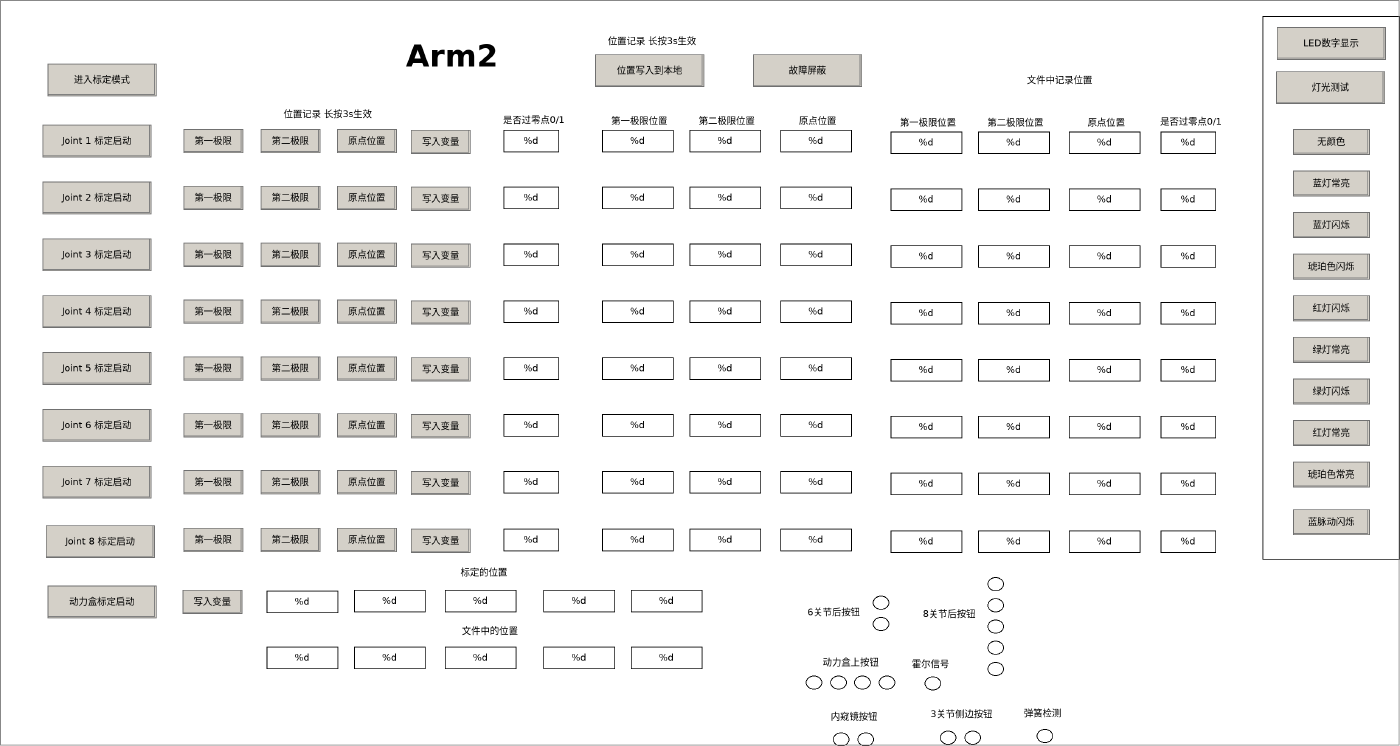
VISUALIZATION arm2Cail  // 1649x879
    Button (56,75 128x38), "进入标定模式", colour toggle: GVL_armCali.g_armEnterCaliMode[2]
        toggle GVL_armCali.g_armEnterCaliMode[2]
    Button (50,147 128x38), "Joint 1 标定启动", colour toggle: GVL_armCali.g_jointIntoCaliState[2][1]
        toggle GVL_armCali.g_jointIntoCaliState[2][1]
    Label (434,40 197x52), "Arm2"
    Button (50,214 128x38), "Joint 2 标定启动", colour toggle: GVL_armCali.g_jointIntoCaliState[2][2]
        toggle GVL_armCali.g_jointIntoCaliState[2][2]
    Button (216,152 70x28), "第一极限", colour toggle: GVL_armCali.g_linkEncFristCaliTrigger[2][1]
        tap GVL_armCali.g_linkEncFristPosCali[2][1]
    Button (307,152 70x28), "第二极限", colour toggle: GVL_armCali.g_linkEncSecondCaliTrigger[2][1]
        tap GVL_armCali.g_linkEncSecondPosCali[2][1]
    Rectangle (593,153 65x26), "%d", text variable: GVL_armCali.g_linkZeroCrossOrNot[2][1]
    Label (588,130 82x23), "是否过零点0/1"
    Rectangle (709,153 84x26), "%d", text variable: GVL_armCali.g_linkLimitFristPos[2][1]
    Label (712,131 82x23), "第一极限位置"
    Rectangle (812,153 84x26), "%d", text variable: GVL_armCali.g_linkLimitSecondPos[2][1]
    Label (815,131 82x23), "第二极限位置"
    Label (311,123 150x23), "位置记录 长按3s生效"
    Rectangle (919,153 84x26), "%d", text variable: GVL_armCali.g_linkHomePos[2][1]
    Label (922,131 82x23), "原点位置"
    Button (397,152 70x28), "原点位置", colour toggle: GVL_armCali.g_linkEncHomePosCaliTrigger[2][1]
        tap GVL_armCali.g_linkEncHomePosCali[2][1]
    Button (701,64 128x38), "位置写入到本地", colour toggle: GVL_armCali.g_caliDataWriteTrigger[2]
        tap GVL_armCali.g_caliDataWrite[2]
    Label (693,37 150x23), "位置记录 长按3s生效"
    Button (216,219 70x28), "第一极限", colour toggle: GVL_armCali.g_linkEncFristCaliTrigger[2][2]
        tap GVL_armCali.g_linkEncFristPosCali[2][2]
    Button (307,219 70x28), "第二极限", colour toggle: GVL_armCali.g_linkEncSecondCaliTrigger[2][2]
        tap GVL_armCali.g_linkEncSecondPosCali[2][2]
    Rectangle (593,220 65x26), "%d", text variable: GVL_armCali.g_linkZeroCrossOrNot[2][2]
    Rectangle (709,220 84x26), "%d", text variable: GVL_armCali.g_linkLimitFristPos[2][2]
    Rectangle (812,220 84x26), "%d", text variable: GVL_armCali.g_linkLimitSecondPos[2][2]
    Rectangle (919,220 84x26), "%d", text variable: GVL_armCali.g_linkHomePos[2][2]
    Button (397,219 70x28), "原点位置", colour toggle: GVL_armCali.g_linkEncHomePosCaliTrigger[2][2]
        tap GVL_armCali.g_linkEncHomePosCali[2][2]
    Button (50,281 128x38), "Joint 3 标定启动", colour toggle: GVL_armCali.g_jointIntoCaliState[2][3]
        toggle GVL_armCali.g_jointIntoCaliState[2][3]
    Button (216,286 70x28), "第一极限", colour toggle: GVL_armCali.g_linkEncFristCaliTrigger[2][3]
        tap GVL_armCali.g_linkEncFristPosCali[2][3]
    Button (307,286 70x28), "第二极限", colour toggle: GVL_armCali.g_linkEncSecondCaliTrigger[2][3]
        tap GVL_armCali.g_linkEncSecondPosCali[2][3]
    Rectangle (593,287 65x26), "%d", text variable: GVL_armCali.g_linkZeroCrossOrNot[2][3]
    Rectangle (709,287 84x26), "%d", text variable: GVL_armCali.g_linkLimitFristPos[2][3]
    Rectangle (812,287 84x26), "%d", text variable: GVL_armCali.g_linkLimitSecondPos[2][3]
    Rectangle (919,287 84x26), "%d", text variable: GVL_armCali.g_linkHomePos[2][3]
    Button (397,286 70x28), "原点位置", colour toggle: GVL_armCali.g_linkEncHomePosCaliTrigger[2][3]
        tap GVL_armCali.g_linkEncHomePosCali[2][3]
    Button (50,348 128x38), "Joint 4 标定启动", colour toggle: GVL_armCali.g_jointIntoCaliState[2][4]
        toggle GVL_armCali.g_jointIntoCaliState[2][4]
    Button (216,353 70x28), "第一极限", colour toggle: GVL_armCali.g_linkEncFristCaliTrigger[2][4]
        tap GVL_armCali.g_linkEncFristPosCali[2][4]
    Button (307,353 70x28), "第二极限", colour toggle: GVL_armCali.g_linkEncSecondCaliTrigger[2][4]
        tap GVL_armCali.g_linkEncSecondPosCali[2][4]
    Rectangle (593,354 65x26), "%d", text variable: GVL_armCali.g_linkZeroCrossOrNot[2][4]
    Rectangle (709,354 84x26), "%d", text variable: GVL_armCali.g_linkLimitFristPos[2][4]
    Rectangle (812,354 84x26), "%d", text variable: GVL_armCali.g_linkLimitSecondPos[2][4]
    Rectangle (919,354 84x26), "%d", text variable: GVL_armCali.g_linkHomePos[2][4]
    Button (397,353 70x28), "原点位置", colour toggle: GVL_armCali.g_linkEncHomePosCaliTrigger[2][4]
        tap GVL_armCali.g_linkEncHomePosCali[2][4]
    Button (50,415 128x38), "Joint 5 标定启动", colour toggle: GVL_armCali.g_jointIntoCaliState[2][5]
        toggle GVL_armCali.g_jointIntoCaliState[2][5]
    Button (216,420 70x28), "第一极限", colour toggle: GVL_armCali.g_linkEncFristCaliTrigger[2][5]
        tap GVL_armCali.g_linkEncFristPosCali[2][5]
    Button (307,420 70x28), "第二极限", colour toggle: GVL_armCali.g_linkEncSecondCaliTrigger[2][5]
        tap GVL_armCali.g_linkEncSecondPosCali[2][5]
    Rectangle (593,421 65x26), "%d", text variable: GVL_armCali.g_linkZeroCrossOrNot[2][5]
    Rectangle (709,421 84x26), "%d", text variable: GVL_armCali.g_linkLimitFristPos[2][5]
    Rectangle (812,421 84x26), "%d", text variable: GVL_armCali.g_linkLimitSecondPos[2][5]
    Rectangle (919,421 84x26), "%d", text variable: GVL_armCali.g_linkHomePos[2][5]
    Button (397,420 70x28), "原点位置", colour toggle: GVL_armCali.g_linkEncHomePosCaliTrigger[2][5]
        tap GVL_armCali.g_linkEncHomePosCali[2][5]
    Button (50,482 128x38), "Joint 6 标定启动", colour toggle: GVL_armCali.g_jointIntoCaliState[2][6]
        toggle GVL_armCali.g_jointIntoCaliState[2][6]
    Button (216,487 70x28), "第一极限", colour toggle: GVL_armCali.g_linkEncFristCaliTrigger[2][6]
        tap GVL_armCali.g_linkEncFristPosCali[2][6]
    Button (307,487 70x28), "第二极限", colour toggle: GVL_armCali.g_linkEncSecondCaliTrigger[2][6]
        tap GVL_armCali.g_linkEncSecondPosCali[2][6]
    Rectangle (593,488 65x26), "%d", text variable: GVL_armCali.g_linkZeroCrossOrNot[2][6]
    Rectangle (709,488 84x26), "%d", text variable: GVL_armCali.g_linkLimitFristPos[2][6]
    Rectangle (812,488 84x26), "%d", text variable: GVL_armCali.g_linkLimitSecondPos[2][6]
    Rectangle (919,488 84x26), "%d", text variable: GVL_armCali.g_linkHomePos[2][6]
    Button (397,487 70x28), "原点位置", colour toggle: GVL_armCali.g_linkEncHomePosCaliTrigger[2][6]
        tap GVL_armCali.g_linkEncHomePosCali[2][6]
    Button (50,549 128x38), "Joint 7 标定启动", colour toggle: GVL_armCali.g_jointIntoCaliState[2][7]
        toggle GVL_armCali.g_jointIntoCaliState[2][7]
    Button (216,554 70x28), "第一极限", colour toggle: GVL_armCali.g_linkEncFristCaliTrigger[2][7]
        tap GVL_armCali.g_linkEncFristPosCali[2][7]
    Button (307,554 70x28), "第二极限", colour toggle: GVL_armCali.g_linkEncSecondCaliTrigger[2][7]
        tap GVL_armCali.g_linkEncSecondPosCali[2][7]
    Rectangle (593,555 65x26), "%d", text variable: GVL_armCali.g_linkZeroCrossOrNot[2][7]
    Rectangle (709,555 84x26), "%d", text variable: GVL_armCali.g_linkLimitFristPos[2][7]
    Rectangle (812,555 84x26), "%d", text variable: GVL_armCali.g_linkLimitSecondPos[2][7]
    Rectangle (919,555 84x26), "%d", text variable: GVL_armCali.g_linkHomePos[2][7]
    Button (397,554 70x28), "原点位置", colour toggle: GVL_armCali.g_linkEncHomePosCaliTrigger[2][7]
        tap GVL_armCali.g_linkEncHomePosCali[2][7]
    Button (54,619 128x38), "Joint 8 标定启动", colour toggle: GVL_armCali.g_jointIntoCaliState[2][8]
        toggle GVL_armCali.g_jointIntoCaliState[2][8]
    Button (216,622 70x28), "第一极限", colour toggle: GVL_armCali.g_linkEncFristCaliTrigger[2][8]
        tap GVL_armCali.g_linkEncFristPosCali[2][8]
    Button (307,622 70x28), "第二极限", colour toggle: GVL_armCali.g_linkEncSecondCaliTrigger[2][8]
        tap GVL_armCali.g_linkEncSecondPosCali[2][8]
    Rectangle (593,623 65x26), "%d", text variable: GVL_armCali.g_linkZeroCrossOrNot[2][8]
    Rectangle (709,623 84x26), "%d", text variable: GVL_armCali.g_linkLimitFristPos[2][8]
    Rectangle (812,623 84x26), "%d", text variable: GVL_armCali.g_linkLimitSecondPos[2][8]
    Rectangle (919,623 84x26), "%d", text variable: GVL_armCali.g_linkHomePos[2][8]
    Button (397,622 70x28), "原点位置", colour toggle: GVL_armCali.g_linkEncHomePosCaliTrigger[2][8]
        tap GVL_armCali.g_linkEncHomePosCali[2][8]
    Rectangle (1049,155 84x26), "%d", text variable: GVL_SetupJointEncoderCaliData.g_minLinkEncoder[2,1]
    Label (1052,133 82x23), "第一极限位置"
    Rectangle (1152,155 84x26), "%d", text variable: GVL_SetupJointEncoderCaliData.g_maxLinkEncoder[2,1]
    Label (1155,133 82x23), "第二极限位置"
    Rectangle (1259,155 84x26), "%d", text variable: GVL_SetupJointEncoderCaliData.g_caliLinkEncoder[2,1]
    Label (1262,133 82x23), "原点位置"
    Rectangle (1049,222 84x26), "%d", text variable: GVL_SetupJointEncoderCaliData.g_minLinkEncoder[2,2]
    Rectangle (1152,222 84x26), "%d", text variable: GVL_SetupJointEncoderCaliData.g_maxLinkEncoder[2,2]
    Rectangle (1259,222 84x26), "%d", text variable: GVL_SetupJointEncoderCaliData.g_caliLinkEncoder[2,2]
    Rectangle (1049,289 84x26), "%d", text variable: GVL_SetupJointEncoderCaliData.g_minLinkEncoder[2,3]
    Rectangle (1152,289 84x26), "%d", text variable: GVL_SetupJointEncoderCaliData.g_maxLinkEncoder[2,3]
    Rectangle (1259,289 84x26), "%d", text variable: GVL_SetupJointEncoderCaliData.g_caliLinkEncoder[2,3]
    Rectangle (1049,356 84x26), "%d", text variable: GVL_SetupJointEncoderCaliData.g_minLinkEncoder[2,4]
    Rectangle (1152,356 84x26), "%d", text variable: GVL_SetupJointEncoderCaliData.g_maxLinkEncoder[2,4]
    Rectangle (1259,356 84x26), "%d", text variable: GVL_SetupJointEncoderCaliData.g_caliLinkEncoder[2,4]
    Rectangle (1049,423 84x26), "%d", text variable: GVL_SetupJointEncoderCaliData.g_minLinkEncoder[2,5]
    Rectangle (1152,423 84x26), "%d", text variable: GVL_SetupJointEncoderCaliData.g_maxLinkEncoder[2,5]
    Rectangle (1259,423 84x26), "%d", text variable: GVL_SetupJointEncoderCaliData.g_caliLinkEncoder[2,5]
    Rectangle (1049,490 84x26), "%d", text variable: GVL_SlaveJointEncoderCaliData.g_minLinkEncoder[2,1]
    Rectangle (1152,490 84x26), "%d", text variable: GVL_SlaveJointEncoderCaliData.g_maxLinkEncoder[2,1]
    Rectangle (1259,490 84x26), "%d", text variable: GVL_SlaveJointEncoderCaliData.g_caliLinkEncoder[2,1]
    Rectangle (1049,557 84x26), "%d", text variable: GVL_SlaveJointEncoderCaliData.g_minLinkEncoder[2,2]
    Rectangle (1152,557 84x26), "%d", text variable: GVL_SlaveJointEncoderCaliData.g_maxLinkEncoder[2,2]
    Rectangle (1259,557 84x26), "%d", text variable: GVL_SlaveJointEncoderCaliData.g_caliLinkEncoder[2,2]
    Rectangle (1049,625 84x26), "%d", text variable: GVL_SlaveJointEncoderCaliData.g_minLinkEncoder[2,3]
    Rectangle (1152,625 84x26), "%d", text variable: GVL_SlaveJointEncoderCaliData.g_maxLinkEncoder[2,3]
    Rectangle (1259,625 84x26), "%d", text variable: GVL_SlaveJointEncoderCaliData.g_caliLinkEncoder[2,3]
    Label (1173,83 150x23), "文件中记录位置"
    Rectangle (1367,155 65x26), "%d", text variable: GVL_SetupJointEncoderCaliData.g_linkEncZeroCross[2,1]
    Label (1362,132 82x23), "是否过零点0/1"
    Rectangle (1367,222 65x26), "%d", text variable: GVL_SetupJointEncoderCaliData.g_linkEncZeroCross[2,2]
    Rectangle (1367,289 65x26), "%d", text variable: GVL_SetupJointEncoderCaliData.g_linkEncZeroCross[2,3]
    Rectangle (1367,356 65x26), "%d", text variable: GVL_SetupJointEncoderCaliData.g_linkEncZeroCross[2,4]
    Rectangle (1367,423 65x26), "%d", text variable: GVL_SetupJointEncoderCaliData.g_linkEncZeroCross[2,5]
    Rectangle (1367,490 65x26), "%d", text variable: GVL_SlaveJointEncoderCaliData.g_linkEncZeroCross[2,1]
    Rectangle (1367,557 65x26), "%d", text variable: GVL_SlaveJointEncoderCaliData.g_linkEncZeroCross[2,2]
    Rectangle (1367,625 65x26), "%d", text variable: GVL_SlaveJointEncoderCaliData.g_linkEncZeroCross[2,3]
    Button (484,153 70x28), "写入变量", colour toggle: GVL_armCali.g_linkPosWriteCaliDataTrigger[2][1]
        tap GVL_armCali.g_linkPosWriteCaliData[2][1]
    Button (484,220 70x28), "写入变量", colour toggle: GVL_armCali.g_linkPosWriteCaliDataTrigger[2][2]
        tap GVL_armCali.g_linkPosWriteCaliData[2][2]
    Button (484,287 70x28), "写入变量", colour toggle: GVL_armCali.g_linkPosWriteCaliDataTrigger[2][3]
        tap GVL_armCali.g_linkPosWriteCaliData[2][3]
    Button (484,354 70x28), "写入变量", colour toggle: GVL_armCali.g_linkPosWriteCaliDataTrigger[2][4]
        tap GVL_armCali.g_linkPosWriteCaliData[2][4]
    Button (484,421 70x28), "写入变量", colour toggle: GVL_armCali.g_linkPosWriteCaliDataTrigger[2][5]
        tap GVL_armCali.g_linkPosWriteCaliData[2][5]
    Button (484,488 70x28), "写入变量", colour toggle: GVL_armCali.g_linkPosWriteCaliDataTrigger[2][6]
        tap GVL_armCali.g_linkPosWriteCaliData[2][6]
    Button (484,555 70x28), "写入变量", colour toggle: GVL_armCali.g_linkPosWriteCaliDataTrigger[2][7]
        tap GVL_armCali.g_linkPosWriteCaliData[2][7]
    Button (484,623 70x28), "写入变量", colour toggle: GVL_armCali.g_linkPosWriteCaliDataTrigger[2][8]
        tap GVL_armCali.g_linkPosWriteCaliData[2][8]
    Button (56,690 128x38), "动力盒标定启动", colour toggle: GVL_armCali.g_powerBoxCali[2]
        toggle GVL_armCali.g_powerBoxCali[2]
    Button (215,695 70x28), "写入变量", colour toggle: GVL_armCali.g_powerBoxPosWriteTrigger[2]
        tap GVL_armCali.g_powerBoxPosWrite[2]
    Rectangle (314,696 84x26), "%d", text variable: GVL_armCali.g_powerBoxLinkHomePos[2][1]
    Rectangle (417,695 84x26), "%d", text variable: GVL_armCali.g_powerBoxLinkHomePos[2][2]
    Rectangle (524,695 84x26), "%d", text variable: GVL_armCali.g_powerBoxLinkHomePos[2][3]
    Rectangle (640,695 84x26), "%d", text variable: GVL_armCali.g_powerBoxLinkHomePos[2][4]
    Rectangle (743,695 84x26), "%d", text variable: GVL_armCali.g_powerBoxLinkHomePos[2][5]
    Rectangle (314,762 84x26), "%d", text variable: GVL_SlaveJointEncoderCaliData.g_caliLinkEncoder[2,4]
    Rectangle (417,762 84x26), "%d", text variable: GVL_SlaveJointEncoderCaliData.g_caliLinkEncoder[2,5]
    Rectangle (524,762 84x26), "%d", text variable: GVL_SlaveJointEncoderCaliData.g_caliLinkEncoder[2,6]
    Rectangle (640,762 84x26), "%d", text variable: GVL_SlaveJointEncoderCaliData.g_caliLinkEncoder[2,7]
    Rectangle (743,762 84x26), "%d", text variable: GVL_SlaveJointEncoderCaliData.g_caliLinkEncoder[2,8]
    Label (502,732 150x23), "文件中的位置"
    Label (495,663 150x23), "标定的位置"
    Label (942,710 80x23), "6关节后按钮"
    Ellipse (1028,727 19x16), colour toggle: GVL_IO.g_joint6IO[2][2]
    Ellipse (1028,702 19x16), colour toggle: GVL_IO.g_joint6IO[2][1]
    Label (1078,712 80x23), "8关节后按钮"
    Ellipse (1163,705 19x16), colour toggle: GVL_IO.g_joint8IO[2][2]
    Ellipse (1163,680 19x16), colour toggle: GVL_IO.g_joint8IO[2][1]
    Ellipse (1163,755 19x16), colour toggle: GVL_IO.g_joint8IO[2][4]
    Ellipse (1163,730 19x16), colour toggle: GVL_IO.g_joint8IO[2][3]
    Label (962,769 80x23), "动力盒上按钮"
    Ellipse (949,796 19x16), colour toggle: GVL_IO.g_jointPowerBoxIO[2][1]
    Ellipse (978,796 19x16), colour toggle: GVL_IO.g_jointPowerBoxIO[2][2]
    Ellipse (1006,796 19x16), colour toggle: GVL_IO.g_jointPowerBoxIO[2][3]
    Ellipse (1035,796 19x16), colour toggle: GVL_IO.g_jointPowerBoxIO[2][4]
    Label (966,833 80x23), "内窥镜按钮"
    Ellipse (981,863 19x16), colour toggle: GVL_IO.g_endoscopeSingle[2][1]
    Ellipse (1010,863 19x16), colour toggle: GVL_IO.g_endoscopeSingle[2][2]
    Ellipse (1163,780 19x16), colour toggle: GVL_IO.g_joint8IO[2][5]
    Ellipse (1089,797 19x16), colour toggle: GVL_IO.g_jointPowerBoxIO[2][5]
    Label (1056,771 80x23), "霍尔信号"
    Rectangle (1487,19 162x640)
    Button (1523,152 90x30), "无颜色", colour toggle: GVL_IO.g_armLight_PowerOff[2]
        toggle GVL_IO.g_armLight_PowerOff[2]
    Button (1523,201 90x30), "蓝灯常亮", colour toggle: GVL_IO.g_armLight_BlueOn[2]
        toggle GVL_IO.g_armLight_BlueOn[2]
    Button (1523,250 90x30), "蓝灯闪烁", colour toggle: GVL_IO.g_armLight_BlueBlink[2]
        toggle GVL_IO.g_armLight_BlueBlink[2]
    Button (1523,299 90x30), "琥珀色闪烁", colour toggle: GVL_IO.g_armLight_AmberBlink[2]
        toggle GVL_IO.g_armLight_AmberBlink[2]
    Button (1523,348 90x30), "红灯闪烁", colour toggle: GVL_IO.g_armLight_RedBlink[2]
        toggle GVL_IO.g_armLight_RedBlink[2]
    Button (1523,397 90x30), "绿灯常亮", colour toggle: GVL_IO.g_armLight_GreenOn[2]
        toggle GVL_IO.g_armLight_GreenOn[2]
    Button (1523,446 90x30), "绿灯闪烁", colour toggle: GVL_IO.g_armLight_GreenBlink[2]
        toggle GVL_IO.g_armLight_GreenBlink[2]
    Button (1503,84 128x38), "灯光测试", colour toggle: GVL_IO.g_lightTest[2]
        toggle GVL_IO.g_lightTest[2]
    Button (1523,495 90x30), "红灯常亮", colour toggle: GVL_IO.g_armLight_redOn[2]
        toggle GVL_IO.g_armLight_redOn[2]
    Button (1523,544 90x30), "琥珀色常亮", colour toggle: GVL_IO.g_armLight_AmberOn[2]
        toggle GVL_IO.g_armLight_AmberOn[2]
    Button (1523,600 90x30), "蓝脉动闪烁", colour toggle: GVL_IO.g_armLight_BluePulse[2]
        toggle GVL_IO.g_armLight_BluePulse[2]
    Button (1504,32 128x38), "LED数字显示", colour toggle: GVL_IO.g_LEDValueDisplay[2]
        toggle GVL_IO.g_LEDValueDisplay[2]
    Label (1075,830 115x23), "3关节侧边按钮"
    Ellipse (1107,861 19x16), colour toggle: GVL_IO.g_asepticMegnetCheck[2][1]
    Ellipse (1136,861 19x16), colour toggle: GVL_IO.g_asepticMegnetCheck[2][2]
    Ellipse (1221,859 19x16)
    Label (1188,829 80x23), "弹簧检测"
    Button (887,64 128x38), "故障屏蔽", colour toggle: g_specialSignal.m_faultMask[2]
        toggle g_specialSignal.m_faultMask[2]
END_VISUALIZATION

(* stored: Version 1.1.0.1, ProductVersion 3.1.4024.11
   Visu arm2Cail: Id {58b436d8-3d98-4529-9a1e-cf6d70f6b95e} *)
